// TwinCAT 3 PLC project PLCStudent
// ProgramVersion: 3.1.4022.3
// libraries:
//   Tc2_Standard, * (Beckhoff Automation GmbH)
//   Tc2_System, * (Beckhoff Automation GmbH)
//   Tc3_Module, * (Beckhoff Automation GmbH)
// project tree:
//   / PlcTask.TcTTO (not stored)
//   POUs/ ControlFBD.TcPOU, MAIN.TcPOU

// ---- POUs/ControlFBD.TcPOU
PROGRAM ControlFBD
VAR
	qxLampStarted	AT %Q* : BOOL;
	gxSliderAout 	AT %Q* : BOOL; 
	gxSliderAin 	AT %Q* : BOOL; 
	gxSliderBout 	AT %Q* : BOOL; 
	gxSliderBin 	AT %Q* : BOOL; 
	gxDrillDown 	AT %Q* : BOOL;
	gxDrillUp		AT %Q* : BOOL;
	
	ixButtonStart	AT %I* : BOOL;
	ixButtonStop	AT %I* : BOOL;
	ixSliderAout	AT %I* : BOOL;
	ixSliderAin		AT %I* : BOOL;
	ixSliderBout	AT %I* : BOOL;
	ixSliderBin		AT %I* : BOOL;
	ixDrillUp		AT %I* : BOOL;
	ixDrillDown		AT %I* : BOOL;

END_VAR

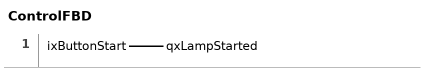
// NETWORK 1
qxLampStarted := ixButtonStart;

END_PROGRAM

// ---- POUs/MAIN.TcPOU
PROGRAM MAIN
VAR
END_VAR

ControlFBD();

END_PROGRAM
